// LS Electric XG5000 project: XGB_Enet02
// PLC NewPLC
// module base 0 slot 0: 입출력 모듈:XBM-DR16S (DC 24V입력, 릴레이 출력 16점)
// module base 0 slot 1: FEnet:XBL-EMTA (Ethernet 통신 모듈, 전기 Master)

PROGRAM NewProgram (task: 스캔 프로그램)

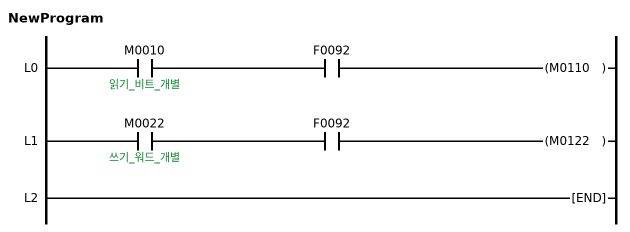
; L0
LOAD      M0010	// 읽기_비트_개별
AND       F0092
OUT       M0110
; L1
LOAD      M0022	// 쓰기_워드_개별
AND       F0092
OUT       M0122
; L2
END

VARIABLES AND COMMENTS (devices not used above)
M00020	BIT	쓰기_비트_개별
M00021	BIT	쓰기_비트_연속
M00023	BIT	쓰기_워드_연속
M00011	BIT	읽기_비트_연속
M00012	BIT	읽기_워드_개별
M00013	BIT	읽기_워드_연속